PROGRAM POU
VAR
	axis : AXIS_REF;
	fbPower : MC_Power;
	fbAbs : MC_MoveAbsolute;
END_VAR

fbPower(
	Axis:= axis, 
	Enable:= , 
	Enable_Positive:= , 
	Enable_Negative:= , 
	Override:= , 
	BufferMode:= , 
	Options:= , 
	Status=> , 
	Busy=> , 
	Active=> , 
	Error=> , 
	ErrorID=> );
	
	fbAbs(
	Axis:= axis, 
	Execute:= , 
	Position:= , 
	Velocity:= , 
	Acceleration:= , 
	Deceleration:= , 
	Jerk:= , 
	BufferMode:= , 
	Options:= , 
	Done=> , 
	Busy=> , 
	Active=> , 
	CommandAborted=> , 
	Error=> , 
	ErrorID=> );

END_PROGRAM

(* stored: Version 1.1.0.1, ProductVersion 3.1.4022.10
   POU POU: Id {7cbb952f-1156-406f-bb5e-e477d1dc07d8}, SpecialFunc None *)
